(* PLC project Device (Win32), 汪勇强测试项目 数学函数指令测试 1 *)
(* stored: creationDateTime 2025-08-30T16:00:00, modificationDateTime 2025-08-30T16:00:00 *)

PROGRAM MathFunctionsTest
  VAR
    Enable : BOOL;
    Complete : BOOL;
    TestValue1 : REAL;  (* UC:[测试输入数据] *)
    TestValue2 : REAL;
    TestValue3 : REAL;
    TestValue4 : REAL;
    TestAngle : REAL;
    ABSResult : REAL;  (* UC:[ABS测试结果] *)
    ACOSResult : REAL;  (* UC:[三角函数测试结果] *)
    ASINResult : REAL;
    ATANResult : REAL;
    COSResult : REAL;
    SINResult : REAL;
    TANResult : REAL;
    EXPResult : REAL;  (* UC:[指数对数函数测试结果] *)
    LNResult : REAL;
    LOGResult : REAL;
    SQRTResult : REAL;  (* UC:[平方根测试结果] *)
    ExpectedReal : REAL;  (* UC:[期望结果变量] *)
    ABSOK : BOOL;  (* UC:[测试结果判断变量] *)
    ACOSOK : BOOL;
    ASINOK : BOOL;
    ATANOG : BOOL;
    COSOK : BOOL;
    SINOK : BOOL;
    TANOG : BOOL;
    EXPOK : BOOL;
    LNOK : BOOL;
    LOGOK : BOOL;
    SQRTOK : BOOL;
    TestStep : INT;  (* UC:[控制变量] *)
    TestsPassed : BOOL;
    Errors : INT;
    Tolerance : REAL;  (* UC:[比较误差容差] *)
    ResultDiff : REAL;
  END_VAR

              Enable := TRUE;
  
  (* 初始化测试数据 *)
  TestValue1 := -5.5;     (* 负数，用于ABS测试 *)
  TestValue2 := 0.5;      (* 0-1之间，用于ACOS/ASIN测试 *)
  TestValue3 := 2.0;      (* 正数，用于指数对数测试 *)
  TestValue4 := 25.0;     (* 完全平方数，用于SQRT测试 *)
  TestAngle := 0.7854;    (* π/4 ≈ 45度，用于三角函数测试 *)
  
  Tolerance := 0.01;      (* 浮点数比较容差 *)

  IF Enable THEN
      
      (* ABS测试 - 绝对值 *)
      TestStep := 1;
      ABSResult := ABS(TestValue1);
      ExpectedReal := 5.5;    (* ABS(-5.5) = 5.5 *)
      ResultDiff := ABSResult - ExpectedReal;
      ABSOK := (ResultDiff < Tolerance) AND (ResultDiff > -Tolerance);
      
      (* ACOS测试 - 反余弦 *)
      TestStep := 2;
      ACOSResult := ACOS(TestValue2);
      ExpectedReal := 1.047;  (* ACOS(0.5) ≈ 1.047弧度 (60度) *)
      ResultDiff := ACOSResult - ExpectedReal;
      ACOSOK := (ResultDiff < Tolerance) AND (ResultDiff > -Tolerance);
      
      (* ASIN测试 - 反正弦 *)
      TestStep := 3;
      ASINResult := ASIN(TestValue2);
      ExpectedReal := 0.524;  (* ASIN(0.5) ≈ 0.524弧度 (30度) *)
      ResultDiff := ASINResult - ExpectedReal;
      ASINOK := (ResultDiff < Tolerance) AND (ResultDiff > -Tolerance);
      
      (* ATAN测试 - 反正切 *)
      TestStep := 4;
      ATANResult := ATAN(1.0);
      ExpectedReal := 0.7854; (* ATAN(1.0) ≈ 0.7854弧度 (45度) *)
      ResultDiff := ATANResult - ExpectedReal;
      ATANOG := (ResultDiff < Tolerance) AND (ResultDiff > -Tolerance);
      
      (* COS测试 - 余弦 *)
      TestStep := 5;
      COSResult := COS(TestAngle);
      ExpectedReal := 0.707;  (* COS(π/4) ≈ 0.707 *)
      ResultDiff := COSResult - ExpectedReal;
      COSOK := (ResultDiff < Tolerance) AND (ResultDiff > -Tolerance);
      
      (* SIN测试 - 正弦 *)
      TestStep := 6;
      SINResult := SIN(TestAngle);
      ExpectedReal := 0.707;  (* SIN(π/4) ≈ 0.707 *)
      ResultDiff := SINResult - ExpectedReal;
      SINOK := (ResultDiff < Tolerance) AND (ResultDiff > -Tolerance);
      
      (* TAN测试 - 正切 *)
      TestStep := 7;
      TANResult := TAN(TestAngle);
      ExpectedReal := 1.0;    (* TAN(π/4) = 1.0 *)
      ResultDiff := TANResult - ExpectedReal;
      TANOG := (ResultDiff < Tolerance) AND (ResultDiff > -Tolerance);
      
      (* EXP测试 - 自然指数 *)
      TestStep := 8;
      EXPResult := EXP(TestValue3);
      ExpectedReal := 7.389;  (* EXP(2.0) ≈ 7.389 *)
      ResultDiff := EXPResult - ExpectedReal;
      EXPOK := (ResultDiff < Tolerance) AND (ResultDiff > -Tolerance);
      
      (* LN测试 - 自然对数 *)
      TestStep := 9;
      LNResult := LN(TestValue3);
      ExpectedReal := 0.693;  (* LN(2.0) ≈ 0.693 *)
      ResultDiff := LNResult - ExpectedReal;
      LNOK := (ResultDiff < Tolerance) AND (ResultDiff > -Tolerance);
      
      (* LOG测试 - 常用对数(以10为底) *)
      TestStep := 10;
      LOGResult := LOG(100.0);
      ExpectedReal := 2.0;    (* LOG(100) = 2.0 *)
      ResultDiff := LOGResult - ExpectedReal;
      LOGOK := (ResultDiff < Tolerance) AND (ResultDiff > -Tolerance);
      
      (* SQRT测试 - 平方根 *)
      TestStep := 11;
      SQRTResult := SQRT(TestValue4);
      ExpectedReal := 5.0;    (* SQRT(25.0) = 5.0 *)
      ResultDiff := SQRTResult - ExpectedReal;
      SQRTOK := (ResultDiff < Tolerance) AND (ResultDiff > -Tolerance);
      
      (* 统计结果 *)
      Errors := 0;
      IF NOT ABSOK THEN Errors := Errors + 1; END_IF;
      IF NOT ACOSOK THEN Errors := Errors + 1; END_IF;
      IF NOT ASINOK THEN Errors := Errors + 1; END_IF;
      IF NOT ATANOG THEN Errors := Errors + 1; END_IF;
      IF NOT COSOK THEN Errors := Errors + 1; END_IF;
      IF NOT SINOK THEN Errors := Errors + 1; END_IF;
      IF NOT TANOG THEN Errors := Errors + 1; END_IF;
      IF NOT EXPOK THEN Errors := Errors + 1; END_IF;
      IF NOT LNOK THEN Errors := Errors + 1; END_IF;
      IF NOT LOGOK THEN Errors := Errors + 1; END_IF;
      IF NOT SQRTOK THEN Errors := Errors + 1; END_IF;
      
      TestsPassed := (Errors = 0);
      Complete := TRUE;
      
      IF TestsPassed THEN
          TestStep := 99;  (* 所有测试通过 *)
      ELSE
          TestStep := 88;  (* 有测试失败 *)
      END_IF;

  ELSE
      TestStep := 0;
      Complete := FALSE;
      TestsPassed := FALSE;
      Errors := 0;
  END_IF;


          
END_PROGRAM

CONFIGURATION config
  RESOURCE resource1 ON PLC
    TASK task0(INTERVAL := T#20ms, PRIORITY := 0);
    PROGRAM instance0 WITH task0 : MathFunctionsTest;
  END_RESOURCE
END_CONFIGURATION
